(* IEC 61131-3 sources: PortalRobot/Portal_robot/Device/application/FB/FB_FAULT_INJECTOR, 9 files *)

(* ---- FB_AXIS_FAULT_INJECTOR.st ---- *)
FUNCTION_BLOCK FB_AXIS_FAULT_INJECTOR
VAR_INPUT
	Request      : ST_AXIS_FAULT_REQUEST; // Запрос тестовой логической ошибки оси
	xOwnerAllowed: BOOL; // Безопасные условия, рассчитанные FB_AXIS
END_VAR
VAR_OUTPUT
	xJogConflict : BOOL; // Одноцикловая пара Jog+ и Jog- для штатной проверки
	Status       : ST_FAULT_INJECTION_STATUS; // Состояние источника для HMI
END_VAR
VAR
	rtJogConflict : R_TRIG; // Фронт команды HMI
END_VAR

// --- BEGIN IMPLEMENTATION ---

rtJogConflict(CLK := Request.xJogConflict);

xJogConflict := FALSE;
Status.xRejected := FALSE;
Status.xAllowed := Request.xEnabled AND xOwnerAllowed;
Status.xBusy := FALSE;
Status.xResetAllowed := FALSE;

IF rtJogConflict.Q THEN
	IF Status.xAllowed THEN
		xJogConflict := TRUE;
	ELSE
		Status.xRejected := TRUE;
		Status.udiRejectSequence := Status.udiRejectSequence + UDINT#1;
		IF Status.udiRejectSequence = UDINT#0 THEN
			Status.udiRejectSequence := UDINT#1;
		END_IF;
	END_IF;
END_IF;

Status.xActive := xJogConflict;

(* ---- FB_AXIS_GROUP_FAULT_INJECTOR.st ---- *)
FUNCTION_BLOCK FB_AXIS_GROUP_FAULT_INJECTOR
VAR_INPUT
	Request       : ST_AXIS_GROUP_FAULT_REQUEST; // Команда диагностической ошибки SM3
	xOwnerAllowed : BOOL; // Безопасные условия, рассчитанные FB_AXIS_GROUP
	xReset        : BOOL; // Штатный сброс группы
	Position      : SMC_POS_REF; // Текущая позиция для команды без перемещения
END_VAR
VAR_OUTPUT
	xError    : BOOL; // Защёлкнутая ошибка тестового Motion FB
	udiErrorID: UDINT; // ErrorID тестового Motion FB
	Status    : ST_FAULT_INJECTION_STATUS; // Состояние источника для HMI
END_VAR
VAR_IN_OUT
	AxisGroup : AXIS_GROUP_REF_SM3; // Ссылка на группу осей SoftMotion
END_VAR
VAR
	fbInvalidMove : MC_MoveDirectAbsolute; // Motion FB с недопустимым параметром
	rtExecute     : R_TRIG; // Фронт запроса HMI
	xExecute      : BOOL; // Execute удерживается до Error или Done
	xErrorLatched : BOOL; // Ошибка хранится до штатного сброса группы
END_VAR

// --- BEGIN IMPLEMENTATION ---

rtExecute(CLK := Request.xExecute);

Status.xRejected := FALSE;
Status.xAllowed := Request.xEnabled AND xOwnerAllowed;

IF xReset THEN
	xExecute := FALSE;
	xErrorLatched := FALSE;
	udiErrorID := UDINT#0;
END_IF;

IF rtExecute.Q THEN
	IF Status.xAllowed THEN
		xExecute := TRUE;
	ELSE
		Status.xRejected := TRUE;
		Status.udiRejectSequence := Status.udiRejectSequence + UDINT#1;
		IF Status.udiRejectSequence = UDINT#0 THEN
			Status.udiRejectSequence := UDINT#1;
		END_IF;
	END_IF;
END_IF;

// По контракту SM3_Robotics VelFactor должен находиться в диапазоне ]0, 1].
// Отрицательное значение формирует Error/ErrorID без принятого перемещения.
fbInvalidMove(
	AxisGroup   := AxisGroup,
	Execute     := xExecute,
	Position    := Position,
	CoordSystem := SMC_COORD_SYSTEM.MCS,
	BufferMode  := MC_BUFFER_MODE.Aborting,
	VelFactor   := -1.0,
	AccFactor   := 1.0,
	JerkFactor  := 1.0
);

IF fbInvalidMove.Error THEN
	xErrorLatched := TRUE;
	udiErrorID := TO_UDINT(fbInvalidMove.ErrorID);
END_IF;

IF fbInvalidMove.Error OR fbInvalidMove.Done THEN
	xExecute := FALSE;
END_IF;

xError := xErrorLatched;
Status.xActive := xErrorLatched;
Status.xBusy := xExecute OR fbInvalidMove.Busy;
Status.xResetAllowed := xErrorLatched AND NOT Status.xBusy;

(* ---- FB_CELL_FAULT_INJECTOR.st ---- *)
FUNCTION_BLOCK FB_CELL_FAULT_INJECTOR
VAR_INPUT
	Request       : ST_CELL_FAULT_REQUEST; // Запрос локальной ошибки менеджера ячейки
	xOwnerAllowed : BOOL; // Безопасные условия, рассчитанные FB_CELL_MANAGER
END_VAR
VAR_OUTPUT
	xBothGrippers : BOOL; // Одноцикловое противоречивое состояние для штатной проверки
	Status        : ST_FAULT_INJECTION_STATUS; // Состояние источника для HMI
END_VAR
VAR
	rtBothGrippers : R_TRIG; // Фронт команды HMI
END_VAR

// --- BEGIN IMPLEMENTATION ---

rtBothGrippers(CLK := Request.xBothGrippers);
xBothGrippers := FALSE;
Status.xRejected := FALSE;
Status.xAllowed := Request.xEnabled AND xOwnerAllowed;
Status.xBusy := FALSE;
Status.xResetAllowed := FALSE;

IF rtBothGrippers.Q THEN
	IF Status.xAllowed THEN
		xBothGrippers := TRUE;
	ELSE
		Status.xRejected := TRUE;
		Status.udiRejectSequence := Status.udiRejectSequence + UDINT#1;
		IF Status.udiRejectSequence = UDINT#0 THEN
			Status.udiRejectSequence := UDINT#1;
		END_IF;
	END_IF;
END_IF;

Status.xActive := xBothGrippers;

(* ---- FB_CELL_SAFETY_FAULT_INJECTOR.st ---- *)
FUNCTION_BLOCK FB_CELL_SAFETY_FAULT_INJECTOR
VAR_INPUT
	Request : ST_CELL_SAFETY_FAULT_REQUEST;
END_VAR
VAR_OUTPUT
	axEmergencyStopStation : ARRAY [1..4] OF BOOL;
	axEmergencyStopCabinet : ARRAY [1..2] OF BOOL;
	xEmergencyStopMpg   : BOOL;
	xPhaseRelayFault    : BOOL;
	xPressureRelayFault : BOOL;
	xSafetyRelayFault   : BOOL;
	axDoorUnlocked      : ARRAY [1..4] OF BOOL;
	Status              : ST_FAULT_INJECTION_STATUS;
END_VAR
VAR
	uiIndex : UINT;
END_VAR

// --- BEGIN IMPLEMENTATION ---

Status.xAllowed := Request.xEnabled;
Status.xBusy := FALSE;
Status.xRejected := FALSE;
Status.xResetAllowed := FALSE;

FOR uiIndex := UINT#1 TO UINT#4 DO
	axEmergencyStopStation[uiIndex] := Request.xEnabled AND Request.axEmergencyStopStation[uiIndex];
	axDoorUnlocked[uiIndex] := Request.xEnabled AND Request.axDoorUnlocked[uiIndex];
END_FOR;
FOR uiIndex := UINT#1 TO UINT#2 DO
	axEmergencyStopCabinet[uiIndex] := Request.xEnabled AND Request.axEmergencyStopCabinet[uiIndex];
END_FOR;
xEmergencyStopMpg := Request.xEnabled AND Request.xEmergencyStopMpg;
xPhaseRelayFault := Request.xEnabled AND Request.xPhaseRelayFault;
xPressureRelayFault := Request.xEnabled AND Request.xPressureRelayFault;
xSafetyRelayFault := Request.xEnabled AND Request.xSafetyRelayFault;

Status.xActive := xEmergencyStopMpg
	OR xPhaseRelayFault
	OR xPressureRelayFault
	OR xSafetyRelayFault;
FOR uiIndex := UINT#1 TO UINT#4 DO
	Status.xActive := Status.xActive
		OR axEmergencyStopStation[uiIndex]
		OR axDoorUnlocked[uiIndex];
END_FOR;
FOR uiIndex := UINT#1 TO UINT#2 DO
	Status.xActive := Status.xActive OR axEmergencyStopCabinet[uiIndex];
END_FOR;

(* ---- FB_GRIPPER_FAULT_INJECTOR.st ---- *)
FUNCTION_BLOCK FB_GRIPPER_FAULT_INJECTOR
VAR_INPUT
	Request       : ST_GRIPPER_FAULT_REQUEST; // Поддерживаемые неисправности захвата
	eActiveAction : E_ROBOT_ACTION; // Текущее действие виртуального захвата
END_VAR
VAR_OUTPUT
	xGripper1Fault : BOOL; // Действующая неисправность первого захвата
	xGripper2Fault : BOOL; // Действующая неисправность второго захвата
	xRotationFault : BOOL; // Действующая неисправность поворота
	xGlobalFault   : BOOL; // Действующая общая неисправность
	xActionFault   : BOOL; // Неисправность относится к текущему действию
	Status         : ST_FAULT_INJECTION_STATUS; // Состояние источника для HMI
END_VAR

// --- BEGIN IMPLEMENTATION ---

xGripper1Fault := Request.xEnabled AND Request.xGripper1Fault;
xGripper2Fault := Request.xEnabled AND Request.xGripper2Fault;
xRotationFault := Request.xEnabled AND Request.xRotationFault;
xGlobalFault := Request.xEnabled AND Request.xGlobalFault;

xActionFault := FALSE;
CASE eActiveAction OF
	E_ROBOT_ACTION.UNCLAMP_1,
	E_ROBOT_ACTION.CLAMP_1:
		xActionFault := xGripper1Fault;

	E_ROBOT_ACTION.UNCLAMP_2,
	E_ROBOT_ACTION.CLAMP_2:
		xActionFault := xGripper2Fault;

	E_ROBOT_ACTION.ROTATE_TO_BLANK,
	E_ROBOT_ACTION.ROTATE_TO_DETAIL:
		xActionFault := xRotationFault;
END_CASE;

Status.xAllowed := Request.xEnabled;
Status.xActive := xGripper1Fault
	OR xGripper2Fault
	OR xRotationFault
	OR xGlobalFault;
Status.xBusy := FALSE;
Status.xResetAllowed := NOT Status.xActive;
Status.xRejected := FALSE;

(* ---- FB_MACHINE_FAULT_INJECTOR.st ---- *)
FUNCTION_BLOCK FB_MACHINE_FAULT_INJECTOR
VAR_INPUT
	Request            : ST_MACHINE_FAULT_REQUEST; // Запросы диагностической инъекции
	MachineStatusRaw    : ST_MACHINE_IO_STATUS; // Неизменённая обратная связь станка
	RobotStatusRaw      : ST_ROBOT_STATUS; // Неизменённая обратная связь робота
	NominalTimeouts     : ST_MACHINE_TIMEOUTS; // Штатные таймауты автомата станка
END_VAR
VAR_OUTPUT
	MachineStatus : ST_MACHINE_IO_STATUS; // Обратная связь, передаваемая FB_MACHINE
	RobotStatus   : ST_ROBOT_STATUS; // Статус робота, передаваемый FB_MACHINE
	Timeouts      : ST_MACHINE_TIMEOUTS; // Действующий профиль таймаутов
	Status        : ST_FAULT_INJECTION_STATUS; // Состояние источника для HMI
END_VAR
VAR CONSTANT
	SIMULATION_TIMEOUT : TIME := T#2S; // Ускоренное время диагностического сценария
END_VAR

// Инжектор не формирует маски ошибок. Он только искажает подтверждения,
// после чего FB_MACHINE обнаруживает штатный TIMEOUT собственными таймерами.

// --- BEGIN IMPLEMENTATION ---

MachineStatus := MachineStatusRaw;
RobotStatus := RobotStatusRaw;
Timeouts := NominalTimeouts;

// Состояние источника аварии не должно оставаться активным после снятия
// соответствующего переключателя. Сам FB_MACHINE при этом сохраняет свою
// защёлкнутую ошибку и сбрасывается отдельной командой из меню станка.
MachineStatus.xAlarm := MachineStatusRaw.xAlarm
	AND Request.xEnabled
	AND (Request.xMachineAlarm OR Request.xDoorFault OR Request.xChuckFault);

Status.xAllowed := Request.xEnabled;
Status.xActive := Request.xEnabled AND (
	Request.xMachineAlarm
	OR Request.xDoorFault
	OR Request.xChuckFault
	OR Request.xTimeoutRobotMove
	OR Request.xTimeoutRobotAction
	OR Request.xTimeoutRobotRelease
	OR Request.xTimeoutDoorOpen
		OR Request.xTimeoutDoorClose
		OR Request.xTimeoutHatchUnlock
	OR Request.xTimeoutChuckOpen
	OR Request.xTimeoutChuckClose
	OR Request.xTimeoutCycleStart
);
Status.xBusy := FALSE;
Status.xResetAllowed := FALSE;
Status.xRejected := FALSE;

IF Request.xEnabled THEN
	IF Request.xTimeoutRobotMove THEN
		RobotStatus.xDone := FALSE;
		Timeouts.tRobotMove := SIMULATION_TIMEOUT;
	END_IF;

	IF Request.xTimeoutRobotAction THEN
		RobotStatus.xDone := FALSE;
		RobotStatus.xGripper1Open := FALSE;
		RobotStatus.xGripper1Closed := FALSE;
		RobotStatus.xGripper2Open := FALSE;
		RobotStatus.xGripper2Closed := FALSE;
		RobotStatus.xRotatedToBlank := FALSE;
		RobotStatus.xRotatedToDetail := FALSE;
		Timeouts.tRobotAction := SIMULATION_TIMEOUT;
	END_IF;

	IF Request.xTimeoutRobotRelease THEN
		RobotStatus.xBusy := TRUE;
		Timeouts.tRobotRelease := SIMULATION_TIMEOUT;
	END_IF;

	IF Request.xTimeoutDoorOpen THEN
		MachineStatus.xDoorOpen := FALSE;
		Timeouts.tDoorOpen := SIMULATION_TIMEOUT;
	END_IF;

	IF Request.xTimeoutDoorClose THEN
		MachineStatus.xDoorClosed := FALSE;
		Timeouts.tDoorClose := SIMULATION_TIMEOUT;
	END_IF;

	IF Request.xTimeoutHatchUnlock THEN
		MachineStatus.xHatchLocked := TRUE;
		Timeouts.tHatchUnlock := SIMULATION_TIMEOUT;
	END_IF;

	IF Request.xTimeoutChuckOpen THEN
		MachineStatus.xChuckUnclamped := FALSE;
		Timeouts.tChuckOpen := SIMULATION_TIMEOUT;
	END_IF;

	IF Request.xTimeoutChuckClose THEN
		MachineStatus.xChuckClamped := FALSE;
		Timeouts.tChuckClose := SIMULATION_TIMEOUT;
	END_IF;

	IF Request.xTimeoutCycleStart THEN
		MachineStatus.xCycleActive := FALSE;
		Timeouts.tCycleStart := SIMULATION_TIMEOUT;
	END_IF;
END_IF;

(* ---- FB_MAGAZINE_FAULT_INJECTOR.st ---- *)
FUNCTION_BLOCK FB_MAGAZINE_FAULT_INJECTOR
VAR_INPUT
	Request       : ST_MAGAZINE_FAULT_REQUEST; // Запросы конкретных ошибок магазина
	xOwnerAllowed : BOOL; // Безопасные условия, рассчитанные FB_MAGAZINE
	xComplete     : BOOL; // Штатная ошибка уже сформирована владельцем
END_VAR
VAR_OUTPUT
	xWrongOperation : BOOL;
	xNoBlank        : BOOL;
	xNoFreeSlot     : BOOL;
	xInvalidSlot    : BOOL;
	xSlotContent    : BOOL;
	xGeometry       : BOOL;
	Status          : ST_FAULT_INJECTION_STATUS; // Состояние источника для HMI
END_VAR
VAR
	rtWrongOperation : R_TRIG;
	rtNoBlank        : R_TRIG;
	rtNoFreeSlot     : R_TRIG;
	rtInvalidSlot    : R_TRIG;
	rtSlotContent    : R_TRIG;
	rtGeometry       : R_TRIG;
	xRequestPulse    : BOOL;
END_VAR

// --- BEGIN IMPLEMENTATION ---

rtWrongOperation(CLK := Request.xWrongOperation);
rtNoBlank(CLK := Request.xNoBlank);
rtNoFreeSlot(CLK := Request.xNoFreeSlot);
rtInvalidSlot(CLK := Request.xInvalidSlot);
rtSlotContent(CLK := Request.xSlotContent);
rtGeometry(CLK := Request.xGeometry);

xRequestPulse := rtWrongOperation.Q
	OR rtNoBlank.Q
	OR rtNoFreeSlot.Q
	OR rtInvalidSlot.Q
	OR rtSlotContent.Q
	OR rtGeometry.Q;

Status.xRejected := FALSE;
Status.xAllowed := Request.xEnabled AND xOwnerAllowed;

IF xComplete THEN
	xWrongOperation := FALSE;
	xNoBlank := FALSE;
	xNoFreeSlot := FALSE;
	xInvalidSlot := FALSE;
	xSlotContent := FALSE;
	xGeometry := FALSE;
END_IF;

IF xRequestPulse THEN
	IF Status.xAllowed THEN
		xWrongOperation := rtWrongOperation.Q;
		xNoBlank := rtNoBlank.Q;
		xNoFreeSlot := rtNoFreeSlot.Q;
		xInvalidSlot := rtInvalidSlot.Q;
		xSlotContent := rtSlotContent.Q;
		xGeometry := rtGeometry.Q;
	ELSE
		Status.xRejected := TRUE;
		Status.udiRejectSequence := Status.udiRejectSequence + UDINT#1;
		IF Status.udiRejectSequence = UDINT#0 THEN
			Status.udiRejectSequence := UDINT#1;
		END_IF;
	END_IF;
END_IF;

Status.xActive := xWrongOperation
	OR xNoBlank
	OR xNoFreeSlot
	OR xInvalidSlot
	OR xSlotContent
	OR xGeometry;
Status.xBusy := Status.xActive;
Status.xResetAllowed := FALSE;

(* ---- FB_POINT_FAULT_INJECTOR.st ---- *)
FUNCTION_BLOCK FB_POINT_FAULT_INJECTOR
VAR_INPUT
	Request       : ST_POINT_FAULT_REQUEST; // Запросы конкретных ошибок точки
	xOwnerAllowed : BOOL; // Безопасные условия, рассчитанные менеджером движения
	xComplete     : BOOL; // Штатная ошибка уже сформирована владельцем
	PointRaw      : ST_POINT; // Исходная корректная точка
END_VAR
VAR_OUTPUT
	Point    : ST_POINT; // Точка, передаваемая штатной проверке
	xExecute : BOOL; // Синтетический запрос проверки без запуска движения
	Status   : ST_FAULT_INJECTION_STATUS; // Состояние источника для HMI
END_VAR
VAR
	rtXOutOfLimit     : R_TRIG;
	rtYOutOfLimit     : R_TRIG;
	rtZOutOfLimit     : R_TRIG;
	rtInvalidVelocity : R_TRIG;
	xRequestPulse     : BOOL;
	xInjectX          : BOOL;
	xInjectY          : BOOL;
	xInjectZ          : BOOL;
	xInjectVelocity   : BOOL;
END_VAR
VAR CONSTANT
	INVALID_COORDINATE : LREAL := 1.0E+09; // Заведомо вне рабочей зоны проверки
END_VAR

// --- BEGIN IMPLEMENTATION ---

rtXOutOfLimit(CLK := Request.xXOutOfLimit);
rtYOutOfLimit(CLK := Request.xYOutOfLimit);
rtZOutOfLimit(CLK := Request.xZOutOfLimit);
rtInvalidVelocity(CLK := Request.xInvalidVelocity);

xRequestPulse := rtXOutOfLimit.Q
	OR rtYOutOfLimit.Q
	OR rtZOutOfLimit.Q
	OR rtInvalidVelocity.Q;

Status.xRejected := FALSE;
Status.xAllowed := Request.xEnabled AND xOwnerAllowed;

IF xComplete THEN
	xInjectX := FALSE;
	xInjectY := FALSE;
	xInjectZ := FALSE;
	xInjectVelocity := FALSE;
END_IF;

IF xRequestPulse THEN
	IF Status.xAllowed THEN
		xInjectX := rtXOutOfLimit.Q;
		xInjectY := rtYOutOfLimit.Q;
		xInjectZ := rtZOutOfLimit.Q;
		xInjectVelocity := rtInvalidVelocity.Q;
	ELSE
		Status.xRejected := TRUE;
		Status.udiRejectSequence := Status.udiRejectSequence + UDINT#1;
		IF Status.udiRejectSequence = UDINT#0 THEN
			Status.udiRejectSequence := UDINT#1;
		END_IF;
	END_IF;
END_IF;

Point := PointRaw;
// Диагностическая инъекция проверяет выбранный дефект, а не состояние
// инженерного хранилища точек.
IF xInjectX OR xInjectY OR xInjectZ OR xInjectVelocity THEN
	Point.xConfigured := TRUE;
END_IF;
IF xInjectX THEN
	Point.X := INVALID_COORDINATE;
END_IF;
IF xInjectY THEN
	Point.Y := INVALID_COORDINATE;
END_IF;
IF xInjectZ THEN
	Point.Z := INVALID_COORDINATE;
END_IF;
IF xInjectVelocity THEN
	Point.SpeedFactor := 0.0;
END_IF;

xExecute := xInjectX OR xInjectY OR xInjectZ OR xInjectVelocity;
Status.xActive := xExecute;
Status.xBusy := xExecute;
Status.xResetAllowed := FALSE;

(* ---- FB_ROBOT_FAULT_INJECTOR.st ---- *)
FUNCTION_BLOCK FB_ROBOT_FAULT_INJECTOR
VAR_INPUT
	Request       : ST_ROBOT_FAULT_REQUEST; // Запросы локальных ошибок робота
	xOwnerAllowed : BOOL; // Безопасные условия, рассчитанные FB_ROBOT
END_VAR
VAR_OUTPUT
	xWrongAction : BOOL; // Одноцикловая недопустимая команда для штатной проверки
	Status       : ST_FAULT_INJECTION_STATUS; // Состояние источника для HMI
END_VAR
VAR
	rtWrongAction : R_TRIG; // Фронт команды HMI
END_VAR

// --- BEGIN IMPLEMENTATION ---

rtWrongAction(CLK := Request.xWrongAction);
xWrongAction := FALSE;
Status.xRejected := FALSE;
Status.xAllowed := Request.xEnabled AND xOwnerAllowed;
Status.xBusy := FALSE;
Status.xResetAllowed := FALSE;

IF rtWrongAction.Q THEN
	IF Status.xAllowed THEN
		xWrongAction := TRUE;
	ELSE
		Status.xRejected := TRUE;
		Status.udiRejectSequence := Status.udiRejectSequence + UDINT#1;
		IF Status.udiRejectSequence = UDINT#0 THEN
			Status.udiRejectSequence := UDINT#1;
		END_IF;
	END_IF;
END_IF;

Status.xActive := xWrongAction;
